{attribute 'GeneratedUsingTerminal: EL1809-0000-0018'}
{attribute addProperty BoxType "EL1809-0000-0018"}
{attribute addProperty Description "EL1809 16Ch. Dig. Input 24V, 3ms"}
{attribute addProperty Physics "KK"}
{attribute addProperty Id "Channel_1AT %I*Channel_830843C11Channel_2AT %I*Channel_830843C11Channel_3AT %I*Channel_830843C11Channel_4AT %I*Channel_830843C11Channel_5AT %I*Channel_830843C11Channel_6AT %I*Channel_830843C11Channel_7AT %I*Channel_830843C11Channel_8AT %I*Channel_830843C11Channel_9AT %I*Channel_830843C11Channel_10AT %I*Channel_830843C11Channel_11AT %I*Channel_830843C11Channel_12AT %I*Channel_830843C11Channel_13AT %I*Channel_830843C11Channel_14AT %I*Channel_830843C11Channel_15AT %I*Channel_830843C11Channel_16AT %I*Channel_830843C11WcStateAT %I*WcState_9091E0EB2InfoDataAT %I*InfoData_6F19DB2B2"}
{attribute addProperty CRC "840269053"}
{attribute addProperty Size "20"}
TYPE EL1809_32157CFD EXTENDS EtcSlaveTerminalBase_947E5A46 :
STRUCT
	{attribute addProperty Name "Channel_1"}
	Channel_1 : Channel_830843C1;
	{attribute addProperty Name "Channel_2"}
	Channel_2 : Channel_830843C1;
	{attribute addProperty Name "Channel_3"}
	Channel_3 : Channel_830843C1;
	{attribute addProperty Name "Channel_4"}
	Channel_4 : Channel_830843C1;
	{attribute addProperty Name "Channel_5"}
	Channel_5 : Channel_830843C1;
	{attribute addProperty Name "Channel_6"}
	Channel_6 : Channel_830843C1;
	{attribute addProperty Name "Channel_7"}
	Channel_7 : Channel_830843C1;
	{attribute addProperty Name "Channel_8"}
	Channel_8 : Channel_830843C1;
	{attribute addProperty Name "Channel_9"}
	Channel_9 : Channel_830843C1;
	{attribute addProperty Name "Channel_10"}
	Channel_10 : Channel_830843C1;
	{attribute addProperty Name "Channel_11"}
	Channel_11 : Channel_830843C1;
	{attribute addProperty Name "Channel_12"}
	Channel_12 : Channel_830843C1;
	{attribute addProperty Name "Channel_13"}
	Channel_13 : Channel_830843C1;
	{attribute addProperty Name "Channel_14"}
	Channel_14 : Channel_830843C1;
	{attribute addProperty Name "Channel_15"}
	Channel_15 : Channel_830843C1;
	{attribute addProperty Name "Channel_16"}
	Channel_16 : Channel_830843C1;
	{attribute addProperty Name "WcState"}
	WcState : WcState_9091E0EB;
	{attribute addProperty Name "InfoData"}
	InfoData : InfoData_6F19DB2B;
END_STRUCT
END_TYPE

(* stored: Version 1.2.0.0, ProductVersion 3.1.4024.9
   DUT EL1809_32157CFD: Id {4f8f6544-ea20-47d5-b00d-764b46b775ad} *)
